FUNCTION_BLOCK ProductOrder_HMI (* Service Interface Function Block Type *)
  (* Standard: 61499-2 *)
  (* Version 0.0, 9/23/2018, dmidro, nxtControl GmbH, template *)
  PACKAGE Main;
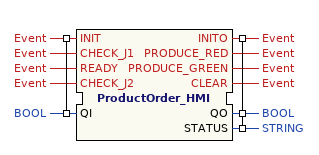
  EVENT_INPUT
    INIT WITH QI;
    CHECK_J1;
    READY;
    CHECK_J2;
  END_EVENT
  EVENT_OUTPUT
    INITO WITH QO, STATUS;
    PRODUCE_RED;
    PRODUCE_GREEN;
    CLEAR;
  END_EVENT
  VAR_INPUT
    QI : BOOL;
  END_VAR
  VAR_OUTPUT
    QO : BOOL; (* Event Output Qualifier *)
    STATUS : STRING; (* Service Status *)
  END_VAR
END_FUNCTION_BLOCK
